ABB RobotStudio station: UiS_E458_nov18.rsstn

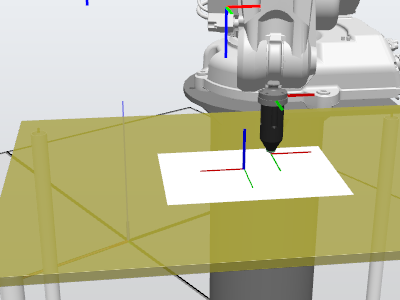
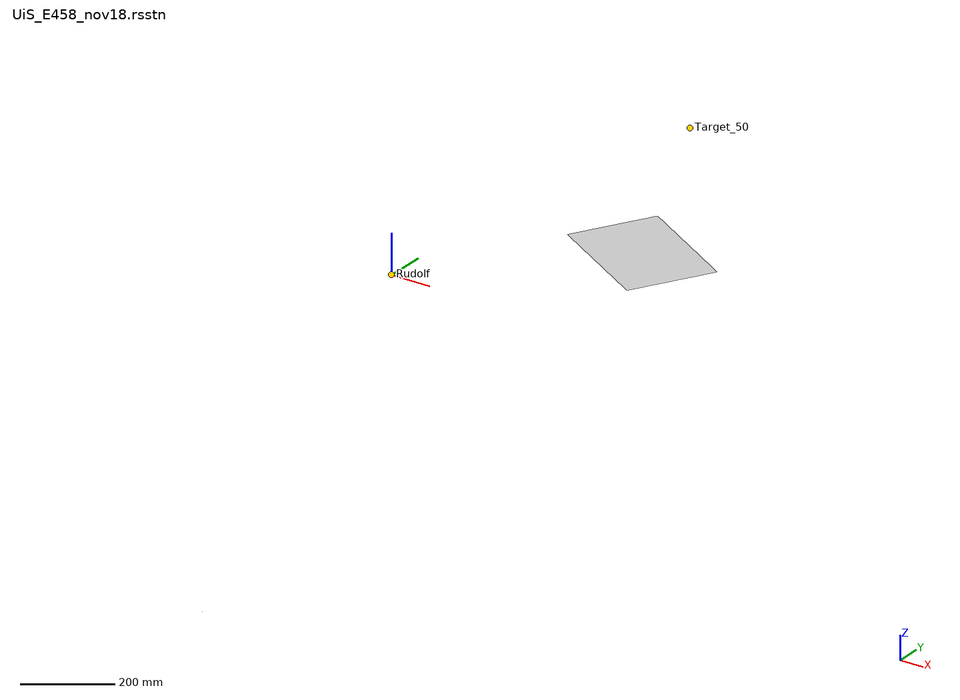
[picture v1: parts stored in the station drawn from their meshes, with robot base, taught points and paths (robot models come from the ABB library and are not in the file)]
Station UiS_E458_nov18 (saved by RobotStudio 25.5.11605.0)
Controller Rudolf, task T_ROB1: task frame (RAPID world) sits at (10, 680, 720) mm, rotated rx 0 ry 0 rz -30 deg in the station
Controller Rudolf
  mechanical unit ROB_1: Rudolf, 6 joints, base frame (0, 0, 0) mm
Layout (positions relative to the parent item):
  - PedestalR [part, from Libraries\Pedestal.rslib] at (10, 680, 0) mm, rotated rx 0 ry 0 rz 150 deg
  - TableR [part, from Libraries\Desk.rslib] at (193.4, 1497.66, 0) mm, rotated rx 0 ry 0 rz -120 deg
  - UISpenholder [mechanism, from Libraries\UISpenholder.rslib] at (307.94, 1016.05, 838.1) mm, rotated rx 180 ry 0 rz 150 deg
  - Rudolf [mechanism, from %ABB.RobotStudio.Models.IRB140%\IRB140_6_81_C_G_03.rslib] at (10, 680, 720) mm, rotated rx 0 ry 0 rz -30 deg; joint values [1.369, 0.9741, 0.381, 0, 0.2157, 1.369] (rad or m)
  - A4sheet [part] at (209.9, 1038.01, 728.1) mm, rotated rx 0 ry 0 rz -30 deg, size 297 x 210 x 0 mm
Attachment: TableR is attached to PedestalR
Attachment: UISpenholder is attached to Rudolf / Link6
Station signals: DI doClose, DI doOpen
Station logic (signal -> signal, property => property):
  Norbert.doOpen -> SC_Gripper.diOpen
  Norbert.doClose -> SC_Gripper.diClose
  SC_Gripper.doClosed -> Norbert.diClosed
Targets, tools, work objects and paths stored in the station, written as RAPID:
! task T_ROB1
MODULE E458PenTest
  PERS tooldata tSimplePen:=[TRUE,[[0,0,110],[1,0,0,0]],[1,[0,0,1],[1,0,0,0],0,0,0]];
  TASK PERS wobjdata wobjTableR:=[FALSE,TRUE,"",[[150,500,8],[1,0,0,0]],[[0,0,0],[1,0,0,0]]];
  CONST robtarget Target_50:=[[50,100,300],[0,0,1,0],[0,0,0,0],[9E+09,9E+09,9E+09,9E+09,9E+09,9E+09]];
  PROC main()
    Path_10;
  ENDPROC
  PROC Path_10()
    MoveL Target_50,v500,z10,tSimplePen\WObj:=wobjTableR;
    MoveL Target_50,v500,z10,tSimplePen\WObj:=wobjTableR;
  ENDPROC
ENDMODULE

! task T_ROB1
MODULE LINKEDM
  PROC Linked_m()
  ENDPROC
ENDMODULE

! task T_ROB1
MODULE E458GripperTest
  CONST robtarget target_K0:=[[0,0,0],[0,1,0,0],[-1,0,0,0],[9E+09,9E+09,9E+09,9E+09,9E+09,9E+09]];
  PROC main()
    MoveL Offs(target_K0, 0, 0, 200),v500,z10,tool0\WObj:=wobj0;
    movePuck;
  ENDPROC
  PROC movePuck()
    MoveJ Offs(target_K0, 0, 0, 200),v500,z10,tool0\WObj:=wobj0;
    WaitTime 1.0;
    MoveJ Offs(target_K0, 0, 0, 200),v500,z10,tool0\WObj:=wobj0;
    WaitTime 1.0;
    MoveJ Offs(target_K0, 0, 0, 200),v500,z10,tool0\WObj:=wobj0;
    WaitTime 1.0;
  ENDPROC
ENDMODULE

! task T_ROB1
MODULE LINKEDM
  PROC Linked_m()
  ENDPROC
ENDMODULE

